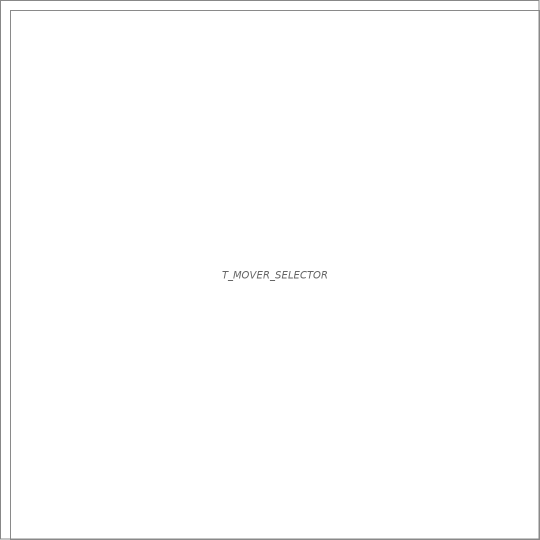
VISUALIZATION SELECTOR_VISU  // 540x540
    Frame (10,10 530x530)
        shows T_MOVER_SELECTOR(Control := GVL_XTS.SelectorCtrl, State := GVL_XTS.SelectorState, sState := MAIN.sSelectorState, sResult := MAIN.sSelectorResult)
END_VISUALIZATION

(* stored: Version 1.1.0.1, ProductVersion 3.1.4026.20
   Visu SELECTOR_VISU: Id {b8157e00-bdc4-41b2-ba88-fc82d6af7c34} *)
